{attribute 'linkalways'} 
{attribute 'no_explicit_call' := 'This FB is a CLASS and must be accessed using methods or properties'}
{attribute 'enable_dynamic_creation'}
FUNCTION_BLOCK QueuedPoolAsyncCommandRunner
VAR
	pool : LinkedList;
	queue : Queue;
	poolCapacity : CollectionSize;
	queueCapacity : CollectionSize;
END_VAR

METHOD PUBLIC CyclicCall
VAR
	enumerator : mobject_collections.I_ForwardEnumerator;
	command : I_AsyncCommand;
END_VAR
IF pool.Count < poolCapacity THEN
	// Need to think about how we handle errors
	IF queue.TryDequeue(command) THEN
		pool.AddLast(command);
		command.Execute();
	END_IF
END_IF

IF pool.Count > 0 THEN
	enumerator := pool.GetEnumerator();
	WHILE enumerator.MoveNext() DO
		IF enumerator.TryGet(command) THEN
			IF command <> 0 THEN
				IF command.Idle THEN
					command.Execute();
				ELSIF command.Executing THEN
					command.CyclicCall();
				ELSIF command.Stopped THEN
					pool.Remove(command);
				END_IF
			END_IF
		END_IF
	END_WHILE
	enumerator.Dispose();
END_IF
END_METHOD

METHOD FB_init : BOOL
VAR_INPUT
	bInitRetains : BOOL; // if TRUE, the retain variables are initialized (warm start / cold start)
	bInCopyCode : BOOL;  // if TRUE, the instance afterwards gets moved into the copy code (online change)
	poolCapacity : CollectionSize; // DINT(1..2147483647)
	queueCapacity : CollectionSize;
END_VAR
THIS^.poolCapacity := poolCapacity;
THIS^.queueCapacity := queueCapacity;
END_METHOD

{attribute 'monitoring' := 'call'}
PROPERTY PUBLIC PoolCount : DINT
GET // PUBLIC
PoolCount := pool.Count;
END_GET
END_PROPERTY

METHOD PUBLIC QueueCommand : BOOL
VAR_INPUT
	command : I_AsyncCommand;
END_VAR
IF pool.Count < poolCapacity THEN
	pool.AddLast(command);
	QueueCommand := TRUE;
	RETURN;
END_IF

IF queue.Count < queueCapacity THEN
	queue.Enqueue(command);
	QueueCommand := TRUE;
	RETURN;
END_IF
END_METHOD

{attribute 'monitoring' := 'call'}
PROPERTY PUBLIC QueueCount : DINT
GET // PUBLIC
QueueCount := queue.Count;
END_GET
END_PROPERTY

END_FUNCTION_BLOCK

(* stored: Version 1.1.0.1, ProductVersion 3.1.4024.12
   POU QueuedPoolAsyncCommandRunner: Id {3d968788-ea35-45c9-ac1d-1da7e9e9bafb}, SpecialFunc None
   Folder Constructor: Id {ed5565cf-5a56-4fe6-afc3-af8867cab854}
   Folder Properties: Id {c90ce1dd-c8ed-450b-9da0-dbdb395ac42b}
   Method CyclicCall: Id {a3426739-d204-44be-9070-f3ff5b14d543}
   Method FB_init: Id {7bf32926-234b-433b-beeb-461c98b51d5b}
   Property PoolCount: Id {70b113a6-3d29-4bdd-9e14-4ca4868f5f93}
   Get Get: Id {c7d533e4-86db-4724-ba6e-c592693cb426}
   Method QueueCommand: Id {38a72f8d-c1be-4057-afa5-cec55af2bbfd}
   Property QueueCount: Id {4ef39e5d-2ea6-488a-ac43-0b38dbb97090}
   Get Get: Id {6975a982-8b9f-4872-8708-a853a493e2fd} *)
